(* IEC 61131-3 sources: SafePLC-Gen-Evaluation/Evaluation Results/eastman/run_02, 2 files *)

(* ---- io_declarations.st ---- *)
(* ==================================================  *)
(* PLC I/O Variable Declarations — CODESYS 3.5  *)
(* Generated by SafePLC-Gen Multimodal  *)
(* ==================================================  *)

VAR_GLOBAL
    (* --- Analog Inputs ---  *)
    FI_1_Raw                     AT %IW0       : INT := 0;    (* FI-1 — Flow indicator on line P-65, feed inlet   *)
    FI_2_Raw                     AT %IW2       : INT := 0;    (* FI-2 — Flow indicator on line P-53, feed to Col  *)
    FI_3_Raw                     AT %IW4       : INT := 0;    (* FI-3 — Flow indicator on line P-57, side draw f  *)
    TI_1_Raw                     AT %IW6       : INT := 0;    (* TI-1 — Temperature indicator, lower left area o  *)
    TI_4_Raw                     AT %IW8       : INT := 0;    (* TI-4 — Temperature indicator on line P-12, feed  *)
    TI_5_Raw                     AT %IW10      : INT := 0;    (* TI-5 — Temperature indicator on line P-53, feed  *)
    TI_6_Raw                     AT %IW12      : INT := 0;    (* TI-6 — Temperature indicator on line P-47/P-48,  *)
    TI_7_Raw                     AT %IW14      : INT := 0;    (* TI-7 — Temperature indicator on right side, ass  *)
    TI_8_Raw                     AT %IW16      : INT := 0;    (* TI-8 — Temperature indicator on Column 3, upper  *)
    (* --- Analog Outputs ---  *)
    V_3_Out                      AT %QW0       : INT := 0;    (* V-3 — Control valve on line P-28, heavy phase   *)
    V_4_Out                      AT %QW2       : INT := 0;    (* V-4 — Control valve on line P-74/P-12, feed fl  *)
    V_5_Out                      AT %QW4       : INT := 0;    (* V-5 — Control valve on line P-38/P-83, reflux   *)
    V_7_Out                      AT %QW6       : INT := 0;    (* V-7 — Control valve on line P-19, overhead vap  *)
END_VAR

(* ---- generated_code.st ---- *)
(* Generated by SafePLC-Gen Multimodal — CODESYS 3.5 *)
(* IEC 61131-3 Structured Text *)
(* Date: 2026-04-25T12:29:26.352487 *)

PROGRAM DistillationColumnControl

VAR
    FI_1_Raw                     AT %IW0       : INT := 0;
    FI_2_Raw                     AT %IW2       : INT := 0;
    FI_3_Raw                     AT %IW4       : INT := 0;
    TI_1_Raw                     AT %IW6       : INT := 0;
    TI_4_Raw                     AT %IW8       : INT := 0;
    TI_5_Raw                     AT %IW10      : INT := 0;
    TI_6_Raw                     AT %IW12      : INT := 0;
    TI_7_Raw                     AT %IW14      : INT := 0;
    TI_8_Raw                     AT %IW16      : INT := 0;
    V_3_Out                      AT %QW0       : INT := 0;
    V_4_Out                      AT %QW2       : INT := 0;
    V_5_Out                      AT %QW4       : INT := 0;
    V_7_Out                      AT %QW6       : INT := 0;
END_VAR

VAR
    FirstScan                    : BOOL := TRUE;

    FI_1_Scaled                  : REAL := 0.0;
    FI_2_Scaled                  : REAL := 0.0;
    FI_3_Scaled                  : REAL := 0.0;
    TI_1_Scaled                  : REAL := 0.0;
    TI_4_Scaled                  : REAL := 0.0;
    TI_5_Scaled                  : REAL := 0.0;
    TI_6_Scaled                  : REAL := 0.0;
    TI_7_Scaled                  : REAL := 0.0;
    TI_8_Scaled                  : REAL := 0.0;

    FI_1_HH_SP                   : REAL := 900.0;
    FI_1_H_SP                    : REAL := 800.0;
    FI_1_L_SP                    : REAL := 200.0;
    FI_1_LL_SP                   : REAL := 100.0;
    FI_1_Deadband                : REAL := 10.0;
    FI_1_H                       : BOOL := FALSE;
    FI_1_L                       : BOOL := FALSE;
    FI_1_HH_Latch                : SR := (S1 := FALSE, R := FALSE);
    FI_1_LL_Latch                : SR := (S1 := FALSE, R := FALSE);
    FI_1_HH_Ack                  : BOOL := FALSE;
    FI_1_LL_Ack                  : BOOL := FALSE;

    FI_2_HH_SP                   : REAL := 900.0;
    FI_2_H_SP                    : REAL := 800.0;
    FI_2_L_SP                    : REAL := 200.0;
    FI_2_LL_SP                   : REAL := 100.0;
    FI_2_Deadband                : REAL := 10.0;
    FI_2_H                       : BOOL := FALSE;
    FI_2_L                       : BOOL := FALSE;
    FI_2_HH_Latch                : SR := (S1 := FALSE, R := FALSE);
    FI_2_LL_Latch                : SR := (S1 := FALSE, R := FALSE);
    FI_2_HH_Ack                  : BOOL := FALSE;
    FI_2_LL_Ack                  : BOOL := FALSE;

    FI_3_HH_SP                   : REAL := 900.0;
    FI_3_H_SP                    : REAL := 800.0;
    FI_3_L_SP                    : REAL := 200.0;
    FI_3_LL_SP                   : REAL := 100.0;
    FI_3_Deadband                : REAL := 10.0;
    FI_3_H                       : BOOL := FALSE;
    FI_3_L                       : BOOL := FALSE;
    FI_3_HH_Latch                : SR := (S1 := FALSE, R := FALSE);
    FI_3_LL_Latch                : SR := (S1 := FALSE, R := FALSE);
    FI_3_HH_Ack                  : BOOL := FALSE;
    FI_3_LL_Ack                  : BOOL := FALSE;

    TI_1_HH_SP                   : REAL := 180.0;
    TI_1_H_SP                    : REAL := 160.0;
    TI_1_L_SP                    : REAL := 60.0;
    TI_1_LL_SP                   : REAL := 40.0;
    TI_1_Deadband                : REAL := 2.0;
    TI_1_H                       : BOOL := FALSE;
    TI_1_L                       : BOOL := FALSE;
    TI_1_HH_Latch                : SR := (S1 := FALSE, R := FALSE);
    TI_1_LL_Latch                : SR := (S1 := FALSE, R := FALSE);
    TI_1_HH_Ack                  : BOOL := FALSE;
    TI_1_LL_Ack                  : BOOL := FALSE;

    TI_4_HH_SP                   : REAL := 180.0;
    TI_4_H_SP                    : REAL := 160.0;
    TI_4_L_SP                    : REAL := 60.0;
    TI_4_LL_SP                   : REAL := 40.0;
    TI_4_Deadband                : REAL := 2.0;
    TI_4_H                       : BOOL := FALSE;
    TI_4_L                       : BOOL := FALSE;
    TI_4_HH_Latch                : SR := (S1 := FALSE, R := FALSE);
    TI_4_LL_Latch                : SR := (S1 := FALSE, R := FALSE);
    TI_4_HH_Ack                  : BOOL := FALSE;
    TI_4_LL_Ack                  : BOOL := FALSE;

    TI_5_HH_SP                   : REAL := 180.0;
    TI_5_H_SP                    : REAL := 160.0;
    TI_5_L_SP                    : REAL := 60.0;
    TI_5_LL_SP                   : REAL := 40.0;
    TI_5_Deadband                : REAL := 2.0;
    TI_5_H                       : BOOL := FALSE;
    TI_5_L                       : BOOL := FALSE;
    TI_5_HH_Latch                : SR := (S1 := FALSE, R := FALSE);
    TI_5_LL_Latch                : SR := (S1 := FALSE, R := FALSE);
    TI_5_HH_Ack                  : BOOL := FALSE;
    TI_5_LL_Ack                  : BOOL := FALSE;

    TI_6_HH_SP                   : REAL := 180.0;
    TI_6_H_SP                    : REAL := 160.0;
    TI_6_L_SP                    : REAL := 60.0;
    TI_6_LL_SP                   : REAL := 40.0;
    TI_6_Deadband                : REAL := 2.0;
    TI_6_H                       : BOOL := FALSE;
    TI_6_L                       : BOOL := FALSE;
    TI_6_HH_Latch                : SR := (S1 := FALSE, R := FALSE);
    TI_6_LL_Latch                : SR := (S1 := FALSE, R := FALSE);
    TI_6_HH_Ack                  : BOOL := FALSE;
    TI_6_LL_Ack                  : BOOL := FALSE;

    TI_7_HH_SP                   : REAL := 180.0;
    TI_7_H_SP                    : REAL := 160.0;
    TI_7_L_SP                    : REAL := 60.0;
    TI_7_LL_SP                   : REAL := 40.0;
    TI_7_Deadband                : REAL := 2.0;
    TI_7_H                       : BOOL := FALSE;
    TI_7_L                       : BOOL := FALSE;
    TI_7_HH_Latch                : SR := (S1 := FALSE, R := FALSE);
    TI_7_LL_Latch                : SR := (S1 := FALSE, R := FALSE);
    TI_7_HH_Ack                  : BOOL := FALSE;
    TI_7_LL_Ack                  : BOOL := FALSE;

    TI_8_HH_SP                   : REAL := 180.0;
    TI_8_H_SP                    : REAL := 160.0;
    TI_8_L_SP                    : REAL := 60.0;
    TI_8_LL_SP                   : REAL := 40.0;
    TI_8_Deadband                : REAL := 2.0;
    TI_8_H                       : BOOL := FALSE;
    TI_8_L                       : BOOL := FALSE;
    TI_8_HH_Latch                : SR := (S1 := FALSE, R := FALSE);
    TI_8_LL_Latch                : SR := (S1 := FALSE, R := FALSE);
    TI_8_HH_Ack                  : BOOL := FALSE;
    TI_8_LL_Ack                  : BOOL := FALSE;

    FC_4_SP                      : REAL := 500.0;
    FC_4_Kp                      : REAL := 1.2;
    FC_4_Ki                      : REAL := 0.05;
    FC_4_Error                   : REAL := 0.0;
    FC_4_Integral                : REAL := 0.0;
    FC_4_Output                  : REAL := 50.0;

    FC_5_SP                      : REAL := 500.0;
    FC_5_Kp                      : REAL := 1.2;
    FC_5_Ki                      : REAL := 0.05;
    FC_5_Error                   : REAL := 0.0;
    FC_5_Integral                : REAL := 0.0;
    FC_5_Output                  : REAL := 50.0;

    FC_6_SP                      : REAL := 500.0;
    FC_6_Kp                      : REAL := 1.2;
    FC_6_Ki                      : REAL := 0.05;
    FC_6_Error                   : REAL := 0.0;
    FC_6_Integral                : REAL := 0.0;
    FC_6_Output                  : REAL := 50.0;

    LC_1_SP                      : REAL := 50.0;
    LC_1_Scaled                  : REAL := 0.0;
    LC_1_Kp                      : REAL := 1.5;
    LC_1_Ki                      : REAL := 0.03;
    LC_1_Error                   : REAL := 0.0;
    LC_1_Integral                : REAL := 0.0;
    LC_1_Output                  : REAL := 50.0;
    LC_1_HH_SP                   : REAL := 90.0;
    LC_1_H_SP                    : REAL := 80.0;
    LC_1_L_SP                    : REAL := 20.0;
    LC_1_LL_SP                   : REAL := 10.0;
    LC_1_Deadband                : REAL := 1.0;
    LC_1_H                       : BOOL := FALSE;
    LC_1_L                       : BOOL := FALSE;
    LC_1_HH_Latch                : SR := (S1 := FALSE, R := FALSE);
    LC_1_LL_Latch                : SR := (S1 := FALSE, R := FALSE);
    LC_1_HH_Ack                  : BOOL := FALSE;
    LC_1_LL_Ack                  : BOOL := FALSE;

    LC_2_SP                      : REAL := 50.0;
    LC_2_Scaled                  : REAL := 0.0;
    LC_2_Kp                      : REAL := 1.5;
    LC_2_Ki                      : REAL := 0.03;
    LC_2_Error                   : REAL := 0.0;
    LC_2_Integral                : REAL := 0.0;
    LC_2_Output                  : REAL := 50.0;
    LC_2_HH_SP                   : REAL := 90.0;
    LC_2_H_SP                    : REAL := 80.0;
    LC_2_L_SP                    : REAL := 20.0;
    LC_2_LL_SP                   : REAL := 10.0;
    LC_2_Deadband                : REAL := 1.0;
    LC_2_H                       : BOOL := FALSE;
    LC_2_L                       : BOOL := FALSE;
    LC_2_HH_Latch                : SR := (S1 := FALSE, R := FALSE);
    LC_2_LL_Latch                : SR := (S1 := FALSE, R := FALSE);
    LC_2_HH_Ack                  : BOOL := FALSE;
    LC_2_LL_Ack                  : BOOL := FALSE;

    LC_3_SP                      : REAL := 50.0;
    LC_3_Scaled                  : REAL := 0.0;
    LC_3_Kp                      : REAL := 1.5;
    LC_3_Ki                      : REAL := 0.03;
    LC_3_Error                   : REAL := 0.0;
    LC_3_Integral                : REAL := 0.0;
    LC_3_Output                  : REAL := 50.0;
    LC_3_HH_SP                   : REAL := 90.0;
    LC_3_H_SP                    : REAL := 80.0;
    LC_3_L_SP                    : REAL := 20.0;
    LC_3_LL_SP                   : REAL := 10.0;
    LC_3_Deadband                : REAL := 1.0;
    LC_3_H                       : BOOL := FALSE;
    LC_3_L                       : BOOL := FALSE;
    LC_3_HH_Latch                : SR := (S1 := FALSE, R := FALSE);
    LC_3_LL_Latch                : SR := (S1 := FALSE, R := FALSE);
    LC_3_HH_Ack                  : BOOL := FALSE;
    LC_3_LL_Ack                  : BOOL := FALSE;

    PC_2_SP                      : REAL := 5.0;
    PC_2_Scaled                  : REAL := 0.0;
    PC_2_Kp                      : REAL := 2.0;
    PC_2_Ki                      : REAL := 0.04;
    PC_2_Error                   : REAL := 0.0;
    PC_2_Integral                : REAL := 0.0;
    PC_2_Output                  : REAL := 50.0;
    PC_2_HH_SP                   : REAL := 9.0;
    PC_2_H_SP                    : REAL := 8.0;
    PC_2_L_SP                    : REAL := 2.0;
    PC_2_LL_SP                   : REAL := 1.0;
    PC_2_Deadband                : REAL := 0.1;
    PC_2_H                       : BOOL := FALSE;
    PC_2_L                       : BOOL := FALSE;
    PC_2_HH_Latch                : SR := (S1 := FALSE, R := FALSE);
    PC_2_LL_Latch                : SR := (S1 := FALSE, R := FALSE);
    PC_2_HH_Ack                  : BOOL := FALSE;
    PC_2_LL_Ack                  : BOOL := FALSE;

    TC_1_SP                      : REAL := 120.0;
    TC_1_Kp                      : REAL := 1.8;
    TC_1_Ki                      : REAL := 0.02;
    TC_1_Error                   : REAL := 0.0;
    TC_1_Integral                : REAL := 0.0;
    TC_1_Output                  : REAL := 50.0;
    TC_1_HH_SP                   : REAL := 180.0;
    TC_1_H_SP                    : REAL := 160.0;
    TC_1_L_SP                    : REAL := 60.0;
    TC_1_LL_SP                   : REAL := 40.0;
    TC_1_Deadband                : REAL := 2.0;
    TC_1_H                       : BOOL := FALSE;
    TC_1_L                       : BOOL := FALSE;
    TC_1_HH_Latch                : SR := (S1 := FALSE, R := FALSE);
    TC_1_LL_Latch                : SR := (S1 := FALSE, R := FALSE);
    TC_1_HH_Ack                  : BOOL := FALSE;
    TC_1_LL_Ack                  : BOOL := FALSE;

    System_Alarm                 : BOOL := FALSE;
END_VAR

IF FirstScan THEN
    V_3_Out       := 6554;
    V_4_Out       := 6554;
    V_5_Out       := 6554;
    V_7_Out       := 6554;
    FC_4_Integral := 0.0;
    FC_5_Integral := 0.0;
    FC_6_Integral := 0.0;
    LC_1_Integral := 0.0;
    LC_2_Integral := 0.0;
    LC_3_Integral := 0.0;
    PC_2_Integral := 0.0;
    TC_1_Integral := 0.0;
    FirstScan     := FALSE;
    RETURN;
END_IF;

FI_1_Scaled := ((INT_TO_REAL(FI_1_Raw) - 6554.0) / (32767.0 - 6554.0)) * 1000.0;
FI_2_Scaled := ((INT_TO_REAL(FI_2_Raw) - 6554.0) / (32767.0 - 6554.0)) * 1000.0;
FI_3_Scaled := ((INT_TO_REAL(FI_3_Raw) - 6554.0) / (32767.0 - 6554.0)) * 1000.0;
TI_1_Scaled := ((INT_TO_REAL(TI_1_Raw) - 6554.0) / (32767.0 - 6554.0)) * 200.0;
TI_4_Scaled := ((INT_TO_REAL(TI_4_Raw) - 6554.0) / (32767.0 - 6554.0)) * 200.0;
TI_5_Scaled := ((INT_TO_REAL(TI_5_Raw) - 6554.0) / (32767.0 - 6554.0)) * 200.0;
TI_6_Scaled := ((INT_TO_REAL(TI_6_Raw) - 6554.0) / (32767.0 - 6554.0)) * 200.0;
TI_7_Scaled := ((INT_TO_REAL(TI_7_Raw) - 6554.0) / (32767.0 - 6554.0)) * 200.0;
TI_8_Scaled := ((INT_TO_REAL(TI_8_Raw) - 6554.0) / (32767.0 - 6554.0)) * 200.0;

LC_1_Scaled := TI_1_Scaled;
LC_2_Scaled := TI_4_Scaled;
LC_3_Scaled := TI_5_Scaled;
PC_2_Scaled := TI_6_Scaled;

FC_4_Error    := FC_4_SP - FI_2_Scaled;
FC_4_Integral := FC_4_Integral + (FC_4_Ki * FC_4_Error);
IF FC_4_Integral > 100.0 THEN
    FC_4_Integral := 100.0;
ELSIF FC_4_Integral < 0.0 THEN
    FC_4_Integral := 0.0;
END_IF;
FC_4_Output := (FC_4_Kp * FC_4_Error) + FC_4_Integral;
IF FC_4_Output > 100.0 THEN
    FC_4_Output := 100.0;
ELSIF FC_4_Output < 0.0 THEN
    FC_4_Output := 0.0;
END_IF;
V_4_Out := REAL_TO_INT(6554.0 + (FC_4_Output / 100.0) * (32767.0 - 6554.0));

FC_5_Error    := FC_5_SP - FI_3_Scaled;
FC_5_Integral := FC_5_Integral + (FC_5_Ki * FC_5_Error);
IF FC_5_Integral > 100.0 THEN
    FC_5_Integral := 100.0;
ELSIF FC_5_Integral < 0.0 THEN
    FC_5_Integral := 0.0;
END_IF;
FC_5_Output := (FC_5_Kp * FC_5_Error) + FC_5_Integral;
IF FC_5_Output > 100.0 THEN
    FC_5_Output := 100.0;
ELSIF FC_5_Output < 0.0 THEN
    FC_5_Output := 0.0;
END_IF;
V_5_Out := REAL_TO_INT(6554.0 + (FC_5_Output / 100.0) * (32767.0 - 6554.0));

FC_6_Error    := FC_6_SP - FI_1_Scaled;
FC_6_Integral := FC_6_Integral + (FC_6_Ki * FC_6_Error);
IF FC_6_Integral > 100.0 THEN
    FC_6_Integral := 100.0;
ELSIF FC_6_Integral < 0.0 THEN
    FC_6_Integral := 0.0;
END_IF;
FC_6_Output := (FC_6_Kp * FC_6_Error) + FC_6_Integral;
IF FC_6_Output > 100.0 THEN
    FC_6_Output := 100.0;
ELSIF FC_6_Output < 0.0 THEN
    FC_6_Output := 0.0;
END_IF;
V_7_Out := REAL_TO_INT(6554.0 + (FC_6_Output / 100.0) * (32767.0 - 6554.0));

LC_1_Error    := LC_1_SP - LC_1_Scaled;
LC_1_Integral := LC_1_Integral + (LC_1_Ki * LC_1_Error);
IF LC_1_Integral > 100.0 THEN
    LC_1_Integral := 100.0;
ELSIF LC_1_Integral < 0.0 THEN
    LC_1_Integral := 0.0;
END_IF;
LC_1_Output := (LC_1_Kp * LC_1_Error) + LC_1_Integral;
IF LC_1_Output > 100.0 THEN
    LC_1_Output := 100.0;
ELSIF LC_1_Output < 0.0 THEN
    LC_1_Output := 0.0;
END_IF;
V_3_Out := REAL_TO_INT(6554.0 + (LC_1_Output / 100.0) * (32767.0 - 6554.0));

LC_2_Error    := LC_2_SP - LC_2_Scaled;
LC_2_Integral := LC_2_Integral + (LC_2_Ki * LC_2_Error);
IF LC_2_Integral > 100.0 THEN
    LC_2_Integral := 100.0;
ELSIF LC_2_Integral < 0.0 THEN
    LC_2_Integral := 0.0;
END_IF;
LC_2_Output := (LC_2_Kp * LC_2_Error) + LC_2_Integral;
IF LC_2_Output > 100.0 THEN
    LC_2_Output := 100.0;
ELSIF LC_2_Output < 0.0 THEN
    LC_2_Output := 0.0;
END_IF;

LC_3_Error    := LC_3_SP - LC_3_Scaled;
LC_3_Integral := LC_3_Integral + (LC_3_Ki * LC_3_Error);
IF LC_3_Integral > 100.0 THEN
    LC_3_Integral := 100.0;
ELSIF LC_3_Integral < 0.0 THEN
    LC_3_Integral := 0.0;
END_IF;
LC_3_Output := (LC_3_Kp * LC_3_Error) + LC_3_Integral;
IF LC_3_Output > 100.0 THEN
    LC_3_Output := 100.0;
ELSIF LC_3_Output < 0.0 THEN
    LC_3_Output := 0.0;
END_IF;

PC_2_Error    := PC_2_SP - PC_2_Scaled;
PC_2_Integral := PC_2_Integral + (PC_2_Ki * PC_2_Error);
IF PC_2_Integral > 100.0 THEN
    PC_2_Integral := 100.0;
ELSIF PC_2_Integral < 0.0 THEN
    PC_2_Integral := 0.0;
END_IF;
PC_2_Output := (PC_2_Kp * PC_2_Error) + PC_2_Integral;
IF PC_2_Output > 100.0 THEN
    PC_2_Output := 100.0;
ELSIF PC_2_Output < 0.0 THEN
    PC_2_Output := 0.0;
END_IF;

TC_1_Error    := TC_1_SP - TI_7_Scaled;
TC_1_Integral := TC_1_Integral + (TC_1_Ki * TC_1_Error);
IF TC_1_Integral > 100.0 THEN
    TC_1_Integral := 100.0;
ELSIF TC_1_Integral < 0.0 THEN
    TC_1_Integral := 0.0;
END_IF;
TC_1_Output := (TC_1_Kp * TC_1_Error) + TC_1_Integral;
IF TC_1_Output > 100.0 THEN
    TC_1_Output := 100.0;
ELSIF TC_1_Output < 0.0 THEN
    TC_1_Output := 0.0;
END_IF;

IF FI_1_Scaled >= FI_1_HH_SP THEN
    FI_1_HH_Latch(S1 := TRUE, R := FALSE);
ELSIF FI_1_Scaled <= (FI_1_HH_SP - FI_1_Deadband) THEN
    FI_1_HH_Latch(S1 := FALSE, R := FI_1_HH_Ack);
END_IF;
IF FI_1_Scaled >= FI_1_H_SP THEN
    FI_1_H := TRUE;
ELSIF FI_1_Scaled <= (FI_1_H_SP - FI_1_Deadband) THEN
    FI_1_H := FALSE;
END_IF;
IF FI_1_Scaled <= FI_1_L_SP THEN
    FI_1_L := TRUE;
ELSIF FI_1_Scaled >= (FI_1_L_SP + FI_1_Deadband) THEN
    FI_1_L := FALSE;
END_IF;
IF FI_1_Scaled <= FI_1_LL_SP THEN
    FI_1_LL_Latch(S1 := TRUE, R := FALSE);
ELSIF FI_1_Scaled >= (FI_1_LL_SP + FI_1_Deadband) THEN
    FI_1_LL_Latch(S1 := FALSE, R := FI_1_LL_Ack);
END_IF;

IF FI_2_Scaled >= FI_2_HH_SP THEN
    FI_2_HH_Latch(S1 := TRUE, R := FALSE);
ELSIF FI_2_Scaled <= (FI_2_HH_SP - FI_2_Deadband) THEN
    FI_2_HH_Latch(S1 := FALSE, R := FI_2_HH_Ack);
END_IF;
IF FI_2_Scaled >= FI_2_H_SP THEN
    FI_2_H := TRUE;
ELSIF FI_2_Scaled <= (FI_2_H_SP - FI_2_Deadband) THEN
    FI_2_H := FALSE;
END_IF;
IF FI_2_Scaled <= FI_2_L_SP THEN
    FI_2_L := TRUE;
ELSIF FI_2_Scaled >= (FI_2_L_SP + FI_2_Deadband) THEN
    FI_2_L := FALSE;
END_IF;
IF FI_2_Scaled <= FI_2_LL_SP THEN
    FI_2_LL_Latch(S1 := TRUE, R := FALSE);
ELSIF FI_2_Scaled >= (FI_2_LL_SP + FI_2_Deadband) THEN
    FI_2_LL_Latch(S1 := FALSE, R := FI_2_LL_Ack);
END_IF;

IF FI_3_Scaled >= FI_3_HH_SP THEN
    FI_3_HH_Latch(S1 := TRUE, R := FALSE);
ELSIF FI_3_Scaled <= (FI_3_HH_SP - FI_3_Deadband) THEN
    FI_3_HH_Latch(S1 := FALSE, R := FI_3_HH_Ack);
END_IF;
IF FI_3_Scaled >= FI_3_H_SP THEN
    FI_3_H := TRUE;
ELSIF FI_3_Scaled <= (FI_3_H_SP - FI_3_Deadband) THEN
    FI_3_H := FALSE;
END_IF;
IF FI_3_Scaled <= FI_3_L_SP THEN
    FI_3_L := TRUE;
ELSIF FI_3_Scaled >= (FI_3_L_SP + FI_3_Deadband) THEN
    FI_3_L := FALSE;
END_IF;
IF FI_3_Scaled <= FI_3_LL_SP THEN
    FI_3_LL_Latch(S1 := TRUE, R := FALSE);
ELSIF FI_3_Scaled >= (FI_3_LL_SP + FI_3_Deadband) THEN
    FI_3_LL_Latch(S1 := FALSE, R := FI_3_LL_Ack);
END_IF;

IF TI_1_Scaled >= TI_1_HH_SP THEN
    TI_1_HH_Latch(S1 := TRUE, R := FALSE);
ELSIF TI_1_Scaled <= (TI_1_HH_SP - TI_1_Deadband) THEN
    TI_1_HH_Latch(S1 := FALSE, R := TI_1_HH_Ack);
END_IF;
IF TI_1_Scaled >= TI_1_H_SP THEN
    TI_1_H := TRUE;
ELSIF TI_1_Scaled <= (TI_1_H_SP - TI_1_Deadband) THEN
    TI_1_H := FALSE;
END_IF;
IF TI_1_Scaled <= TI_1_L_SP THEN
    TI_1_L := TRUE;
ELSIF TI_1_Scaled >= (TI_1_L_SP + TI_1_Deadband) THEN
    TI_1_L := FALSE;
END_IF;
IF TI_1_Scaled <= TI_1_LL_SP THEN
    TI_1_LL_Latch(S1 := TRUE, R := FALSE);
ELSIF TI_1_Scaled >= (TI_1_LL_SP + TI_1_Deadband) THEN
    TI_1_LL_Latch(S1 := FALSE, R := TI_1_LL_Ack);
END_IF;

IF TI_4_Scaled >= TI_4_HH_SP THEN
    TI_4_HH_Latch(S1 := TRUE, R := FALSE);
ELSIF TI_4_Scaled <= (TI_4_HH_SP - TI_4_Deadband) THEN
    TI_4_HH_Latch(S1 := FALSE, R := TI_4_HH_Ack);
END_IF;
IF TI_4_Scaled >= TI_4_H_SP THEN
    TI_4_H := TRUE;
ELSIF TI_4_Scaled <= (TI_4_H_SP - TI_4_Deadband) THEN
    TI_4_H := FALSE;
END_IF;
IF TI_4_Scaled <= TI_4_L_SP THEN
    TI_4_L := TRUE;
ELSIF TI_4_Scaled >= (TI_4_L_SP + TI_4_Deadband) THEN
    TI_4_L := FALSE;
END_IF;
IF TI_4_Scaled <= TI_4_LL_SP THEN
    TI_4_LL_Latch(S1 := TRUE, R := FALSE);
ELSIF TI_4_Scaled >= (TI_4_LL_SP + TI_4_Deadband) THEN
    TI_4_LL_Latch(S1 := FALSE, R := TI_4_LL_Ack);
END_IF;

IF TI_5_Scaled >= TI_5_HH_SP THEN
    TI_5_HH_Latch(S1 := TRUE, R := FALSE);
ELSIF TI_5_Scaled <= (TI_5_HH_SP - TI_5_Deadband) THEN
    TI_5_HH_Latch(S1 := FALSE, R := TI_5_HH_Ack);
END_IF;
IF TI_5_Scaled >= TI_5_H_SP THEN
    TI_5_H := TRUE;
ELSIF TI_5_Scaled <= (TI_5_H_SP - TI_5_Deadband) THEN
    TI_5_H := FALSE;
END_IF;
IF TI_5_Scaled <= TI_5_L_SP THEN
    TI_5_L := TRUE;
ELSIF TI_5_Scaled >= (TI_5_L_SP + TI_5_Deadband) THEN
    TI_5_L := FALSE;
END_IF;
IF TI_5_Scaled <= TI_5_LL_SP THEN
    TI_5_LL_Latch(S1 := TRUE, R := FALSE);
ELSIF TI_5_Scaled >= (TI_5_LL_SP + TI_5_Deadband) THEN
    TI_5_LL_Latch(S1 := FALSE, R := TI_5_LL_Ack);
END_IF;

IF TI_6_Scaled >= TI_6_HH_SP THEN
    TI_6_HH_Latch(S1 := TRUE, R := FALSE);
ELSIF TI_6_Scaled <= (TI_6_HH_SP - TI_6_Deadband) THEN
    TI_6_HH_Latch(S1 := FALSE, R := TI_6_HH_Ack);
END_IF;
IF TI_6_Scaled >= TI_6_H_SP THEN
    TI_6_H := TRUE;
ELSIF TI_6_Scaled <= (TI_6_H_SP - TI_6_Deadband) THEN
    TI_6_H := FALSE;
END_IF;
IF TI_6_Scaled <= TI_6_L_SP THEN
    TI_6_L := TRUE;
ELSIF TI_6_Scaled >= (TI_6_L_SP + TI_6_Deadband) THEN
    TI_6_L := FALSE;
END_IF;
IF TI_6_Scaled <= TI_6_LL_SP THEN
    TI_6_LL_Latch(S1 := TRUE, R := FALSE);
ELSIF TI_6_Scaled >= (TI_6_LL_SP + TI_6_Deadband) THEN
    TI_6_LL_Latch(S1 := FALSE, R := TI_6_LL_Ack);
END_IF;

IF TI_7_Scaled >= TI_7_HH_SP THEN
    TI_7_HH_Latch(S1 := TRUE, R := FALSE);
ELSIF TI_7_Scaled <= (TI_7_HH_SP - TI_7_Deadband) THEN
    TI_7_HH_Latch(S1 := FALSE, R := TI_7_HH_Ack);
END_IF;
IF TI_7_Scaled >= TI_7_H_SP THEN
    TI_7_H := TRUE;
ELSIF TI_7_Scaled <= (TI_7_H_SP - TI_7_Deadband) THEN
    TI_7_H := FALSE;
END_IF;
IF TI_7_Scaled <= TI_7_L_SP THEN
    TI_7_L := TRUE;
ELSIF TI_7_Scaled >= (TI_7_L_SP + TI_7_Deadband) THEN
    TI_7_L := FALSE;
END_IF;
IF TI_7_Scaled <= TI_7_LL_SP THEN
    TI_7_LL_Latch(S1 := TRUE, R := FALSE);
ELSIF TI_7_Scaled >= (TI_7_LL_SP + TI_7_Deadband) THEN
    TI_7_LL_Latch(S1 := FALSE, R := TI_7_LL_Ack);
END_IF;

IF TI_7_Scaled >= TC_1_HH_SP THEN
    TC_1_HH_Latch(S1 := TRUE, R := FALSE);
ELSIF TI_7_Scaled <= (TC_1_HH_SP - TC_1_Deadband) THEN
    TC_1_HH_Latch(S1 := FALSE, R := TC_1_HH_Ack);
END_IF;
IF TI_7_Scaled >= TC_1_H_SP THEN
    TC_1_H := TRUE;
ELSIF TI_7_Scaled <= (TC_1_H_SP - TC_1_Deadband) THEN
    TC_1_H := FALSE;
END_IF;
IF TI_7_Scaled <= TC_1_L_SP THEN
    TC_1_L := TRUE;
ELSIF TI_7_Scaled >= (TC_1_L_SP + TC_1_Deadband) THEN
    TC_1_L := FALSE;
END_IF;
IF TI_7_Scaled <= TC_1_LL_SP THEN
    TC_1_LL_Latch(S1 := TRUE, R := FALSE);
ELSIF TI_7_Scaled >= (TC_1_LL_SP + TC_1_Deadband) THEN
    TC_1_LL_Latch(S1 := FALSE, R := TC_1_LL_Ack);
END_IF;

IF TI_8_Scaled >= TI_8_HH_SP THEN
    TI_8_HH_Latch(S1 := TRUE, R := FALSE);
ELSIF TI_8_Scaled <= (TI_8_HH_SP - TI_8_Deadband) THEN
    TI_8_HH_Latch(S1 := FALSE, R := TI_8_HH_Ack);
END_IF;
IF TI_8_Scaled >= TI_8_H_SP THEN
    TI_8_H := TRUE;
ELSIF TI_8_Scaled <= (TI_8_H_SP - TI_8_Deadband) THEN
    TI_8_H := FALSE;
END_IF;
IF TI_8_Scaled <= TI_8_L_SP THEN
    TI_8_L := TRUE;
ELSIF TI_8_Scaled >= (TI_8_L_SP + TI_8_Deadband) THEN
    TI_8_L := FALSE;
END_IF;
IF TI_8_Scaled <= TI_8_LL_SP THEN
    TI_8_LL_Latch(S1 := TRUE, R := FALSE);
ELSIF TI_8_Scaled >= (TI_8_LL_SP + TI_8_Deadband) THEN
    TI_8_LL_Latch(S1 := FALSE, R := TI_8_LL_Ack);
END_IF;

IF LC_1_Scaled >= LC_1_HH_SP THEN
    LC_1_HH_Latch(S1 := TRUE, R := FALSE);
ELSIF LC_1_Scaled <= (LC_1_HH_SP - LC_1_Deadband) THEN
    LC_1_HH_Latch(S1 := FALSE, R := LC_1_HH_Ack);
END_IF;
IF LC_1_Scaled >= LC_1_H_SP THEN
    LC_1_H := TRUE;
ELSIF LC_1_Scaled <= (LC_1_H_SP - LC_1_Deadband) THEN
    LC_1_H := FALSE;
END_IF;
IF LC_1_Scaled <= LC_1_L_SP THEN
    LC_1_L := TRUE;
ELSIF LC_1_Scaled >= (LC_1_L_SP + LC_1_Deadband) THEN
    LC_1_L := FALSE;
END_IF;
IF LC_1_Scaled <= LC_1_LL_SP THEN
    LC_1_LL_Latch(S1 := TRUE, R := FALSE);
ELSIF LC_1_Scaled >= (LC_1_LL_SP + LC_1_Deadband) THEN
    LC_1_LL_Latch(S1 := FALSE, R := LC_1_LL_Ack);
END_IF;

IF LC_2_Scaled >= LC_2_HH_SP THEN
    LC_2_HH_Latch(S1 := TRUE, R := FALSE);
ELSIF LC_2_Scaled <= (LC_2_HH_SP - LC_2_Deadband) THEN
    LC_2_HH_Latch(S1 := FALSE, R := LC_2_HH_Ack);
END_IF;
IF LC_2_Scaled >= LC_2_H_SP THEN
    LC_2_H := TRUE;
ELSIF LC_2_Scaled <= (LC_2_H_SP - LC_2_Deadband) THEN
    LC_2_H := FALSE;
END_IF;
IF LC_2_Scaled <= LC_2_L_SP THEN
    LC_2_L := TRUE;
ELSIF LC_2_Scaled >= (LC_2_L_SP + LC_2_Deadband) THEN
    LC_2_L := FALSE;
END_IF;
IF LC_2_Scaled <= LC_2_LL_SP THEN
    LC_2_LL_Latch(S1 := TRUE, R := FALSE);
ELSIF LC_2_Scaled >= (LC_2_LL_SP + LC_2_Deadband) THEN
    LC_2_LL_Latch(S1 := FALSE, R := LC_2_LL_Ack);
END_IF;

IF LC_3_Scaled >= LC_3_HH_SP THEN
    LC_3_HH_Latch(S1 := TRUE, R := FALSE);
ELSIF LC_3_Scaled <= (LC_3_HH_SP - LC_3_Deadband) THEN
    LC_3_HH_Latch(S1 := FALSE, R := LC_3_HH_Ack);
END_IF;
IF LC_3_Scaled >= LC_3_H_SP THEN
    LC_3_H := TRUE;
ELSIF LC_3_Scaled <= (LC_3_H_SP - LC_3_Deadband) THEN
    LC_3_H := FALSE;
END_IF;
IF LC_3_Scaled <= LC_3_L_SP THEN
    LC_3_L := TRUE;
ELSIF LC_3_Scaled >= (LC_3_L_SP + LC_3_Deadband) THEN
    LC_3_L := FALSE;
END_IF;
IF LC_3_Scaled <= LC_3_LL_SP THEN
    LC_3_LL_Latch(S1 := TRUE, R := FALSE);
ELSIF LC_3_Scaled >= (LC_3_LL_SP + LC_3_Deadband) THEN
    LC_3_LL_Latch(S1 := FALSE, R := LC_3_LL_Ack);
END_IF;

IF PC_2_Scaled >= PC_2_HH_SP THEN
    PC_2_HH_Latch(S1 := TRUE, R := FALSE);
ELSIF PC_2_Scaled <= (PC_2_HH_SP - PC_2_Deadband) THEN
    PC_2_HH_Latch(S1 := FALSE, R := PC_2_HH_Ack);
END_IF;
IF PC_2_Scaled >= PC_2_H_SP THEN
    PC_2_H := TRUE;
ELSIF PC_2_Scaled <= (PC_2_H_SP - PC_2_Deadband) THEN
    PC_2_H := FALSE;
END_IF;
IF PC_2_Scaled <= PC_2_L_SP THEN
    PC_2_L := TRUE;
ELSIF PC_2_Scaled >= (PC_2_L_SP + PC_2_Deadband) THEN
    PC_2_L := FALSE;
END_IF;
IF PC_2_Scaled <= PC_2_LL_SP THEN
    PC_2_LL_Latch(S1 := TRUE, R := FALSE);
ELSIF PC_2_Scaled >= (PC_2_LL_SP + PC_2_Deadband) THEN
    PC_2_LL_Latch(S1 := FALSE, R := PC_2_LL_Ack);
END_IF;

System_Alarm :=
    FI_1_HH_Latch.Q1 OR FI_1_LL_Latch.Q1 OR FI_1_H OR FI_1_L OR
    FI_2_HH_Latch.Q1 OR FI_2_LL_Latch.Q1 OR FI_2_H OR FI_2_L OR
    FI_3_HH_Latch.Q1 OR FI_3_LL_Latch.Q1 OR FI_3_H OR FI_3_L OR
    TI_1_HH_Latch.Q1 OR TI_1_LL_Latch.Q1 OR TI_1_H OR TI_1_L OR
    TI_4_HH_Latch.Q1 OR TI_4_LL_Latch.Q1 OR TI_4_H OR TI_4_L OR
    TI_5_HH_Latch.Q1 OR TI_5_LL_Latch.Q1 OR TI_5_H OR TI_5_L OR
    TI_6_HH_Latch.Q1 OR TI_6_LL_Latch.Q1 OR TI_6_H OR TI_6_L OR
    TI_7_HH_Latch.Q1 OR TI_7_LL_Latch.Q1 OR TI_7_H OR TI_7_L OR
    TI_8_HH_Latch.Q1 OR TI_8_LL_Latch.Q1 OR TI_8_H OR TI_8_L OR
    LC_1_HH_Latch.Q1 OR LC_1_LL_Latch.Q1 OR LC_1_H OR LC_1_L OR
    LC_2_HH_Latch.Q1 OR LC_2_LL_Latch.Q1 OR LC_2_H OR LC_2_L OR
    LC_3_HH_Latch.Q1 OR LC_3_LL_Latch.Q1 OR LC_3_H OR LC_3_L OR
    PC_2_HH_Latch.Q1 OR PC_2_LL_Latch.Q1 OR PC_2_H OR PC_2_L OR
    TC_1_HH_Latch.Q1 OR TC_1_LL_Latch.Q1 OR TC_1_H OR TC_1_L;

END_PROGRAM
